// TIA Portal V15.1 export
// export: Created 2024-06-21T08:40:54.1245621Z, ExportSetting WithDefaults, DisplayName Totally Integrated Automation Portal, DisplayVersion V15.1 Update 5, DisplayName TIA Portal Openness, DisplayVersion V15.1 Update 5, DisplayName SINAMICS Startdrive Advanced, DisplayVersion V15.1, DisplayName G130, G150, S120, S150, SINAMICS MV, S210, DisplayVersion V15.1, DisplayName G110M, G120, G120C, G120D, G120P, DisplayVersion V15.1, DisplayName STEP 7 Professional, DisplayVersion V15.1 Update 5, DisplayName STEP 7 Safety, DisplayVersion V15.1, DisplayName WinCC Professional, DisplayVersion V15.1 Update 5, DisplayName SIMATIC Visualization Architect, DisplayVersion V15.1
FUNCTION "LBitToDword" : Void   // FC1027, FBD
TITLE = LBitToDWord
{ S7_Optimized_Access := 'TRUE' }
AUTHOR : VCC
FAMILY : Control
VERSION : 0.1
// =============================================================================
// Handles the conversion from bits to one DWord
// =============================================================================
// stored: AutoNumber false, IsIECCheckEnabled false, SetENOAutomatically False, UDAEnableTagReadback false
   VAR_INPUT
      I_0 : Bool;   // Alarm 00 / Input0
      I_1 : Bool;   // Alarm 01 / Input1
      I_2 : Bool;   // Alarm 02 / Input2
      I_3 : Bool;   // Alarm 03 / Input3
      I_4 : Bool;   // Alarm 04 / Input4
      I_5 : Bool;   // Alarm 05 / Input5
      I_6 : Bool;   // Alarm 06 / Input6
      I_7 : Bool;   // Alarm 07 / Input7
      I_8 : Bool;   // Alarm 08 / Input8
      I_9 : Bool;   // Alarm 09 / Input9
      I_10 : Bool;   // Alarm 10 / Input10
      I_11 : Bool;   // Alarm 11 / Input11
      I_12 : Bool;   // Alarm 12 / Input12
      I_13 : Bool;   // Alarm 13 / Input13
      I_14 : Bool;   // Alarm 14 / Input14
      I_15 : Bool;   // Alarm 15 / Input15
      I_16 : Bool;   // Alarm16 / Input16
      I_17 : Bool;   // Alarm17 / Input17
      I_18 : Bool;   // Alarm18 / Input18
      I_19 : Bool;   // Alarm19 / Input19
      I_20 : Bool;   // Alarm20 / Input20
      I_21 : Bool;   // Alarm21 / Input21
      I_22 : Bool;   // Alarm22 / Input22
      I_23 : Bool;   // Alarm23 / Input23
      I_24 : Bool;   // Alarm24 / Input24
      I_25 : Bool;   // Alarm25 / Input25
      I_26 : Bool;   // Alarm26 / Input26
      I_27 : Bool;   // Alarm27 / Input27
      I_28 : Bool;   // Alarm28 / Input28
      I_29 : Bool;   // Alarm29 / Input29
      I_30 : Bool;   // Alarm30 / Input30
      I_31 : Bool;   // Alarm31 / Input31
   END_VAR
   VAR_OUTPUT
      O_DWord : DWord;   // Alarn DWord for HMI / Dword Out
   END_VAR
BEGIN

REGION Network 1: Temp variable for HMI animation / **** 1 - Inputs **** Move Bit to temporary Word
   // Input
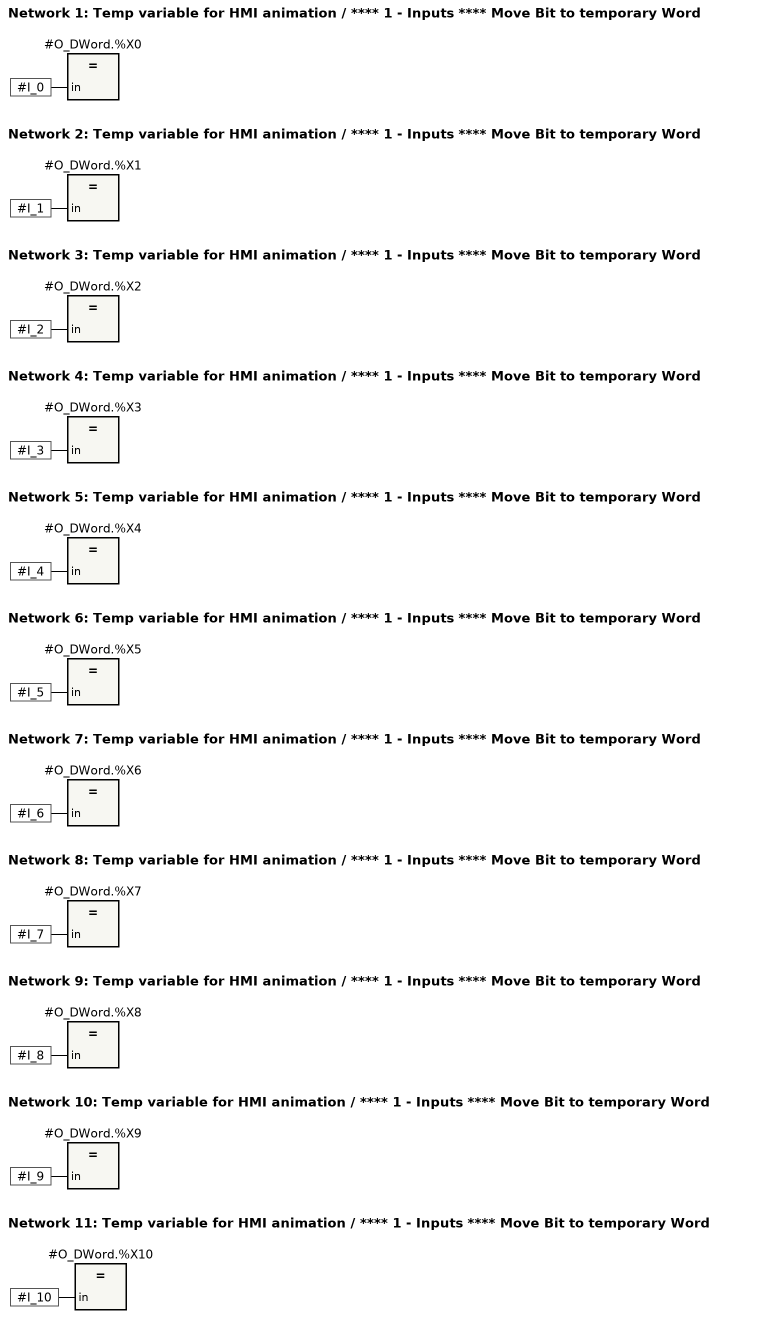
   #O_DWord.%X0 := #I_0;
END_REGION

REGION Network 2: Temp variable for HMI animation / **** 1 - Inputs **** Move Bit to temporary Word
   // Input
   #O_DWord.%X1 := #I_1;
END_REGION

REGION Network 3: Temp variable for HMI animation / **** 1 - Inputs **** Move Bit to temporary Word
   // Input
   #O_DWord.%X2 := #I_2;
END_REGION

REGION Network 4: Temp variable for HMI animation / **** 1 - Inputs **** Move Bit to temporary Word
   // Input
   #O_DWord.%X3 := #I_3;
END_REGION

REGION Network 5: Temp variable for HMI animation / **** 1 - Inputs **** Move Bit to temporary Word
   // Input
   #O_DWord.%X4 := #I_4;
END_REGION

REGION Network 6: Temp variable for HMI animation / **** 1 - Inputs **** Move Bit to temporary Word
   // Input
   #O_DWord.%X5 := #I_5;
END_REGION

REGION Network 7: Temp variable for HMI animation / **** 1 - Inputs **** Move Bit to temporary Word
   // Input
   #O_DWord.%X6 := #I_6;
END_REGION

REGION Network 8: Temp variable for HMI animation / **** 1 - Inputs **** Move Bit to temporary Word
   #O_DWord.%X7 := #I_7;
END_REGION

REGION Network 9: Temp variable for HMI animation / **** 1 - Inputs **** Move Bit to temporary Word
   // Input
   #O_DWord.%X8 := #I_8;
END_REGION

REGION Network 10: Temp variable for HMI animation / **** 1 - Inputs **** Move Bit to temporary Word
   // Input
   #O_DWord.%X9 := #I_9;
END_REGION

REGION Network 11: Temp variable for HMI animation / **** 1 - Inputs **** Move Bit to temporary Word
   // Input
   #O_DWord.%X10 := #I_10;
END_REGION

REGION Network 12: Temp variable for HMI animation / **** 1 - Inputs **** Move Bit to temporary Word
   // Input
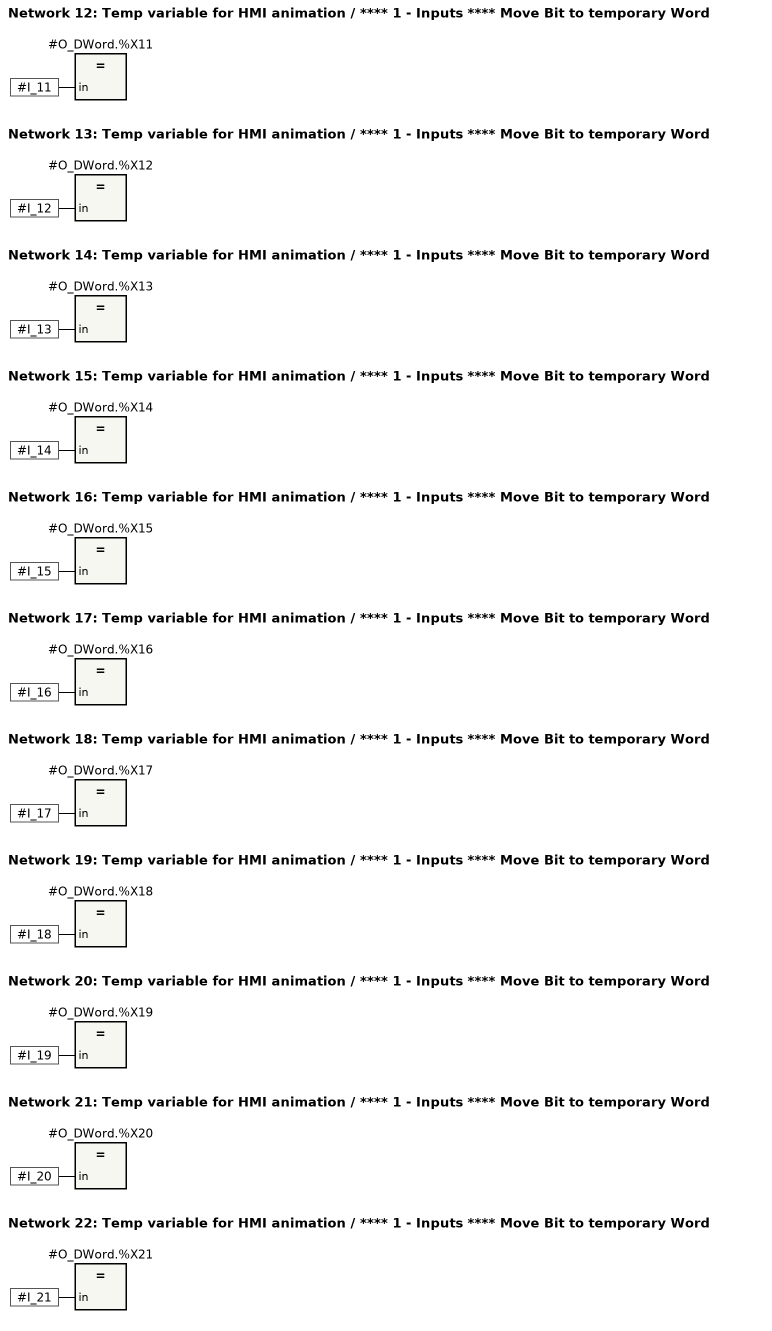
   #O_DWord.%X11 := #I_11;
END_REGION

REGION Network 13: Temp variable for HMI animation / **** 1 - Inputs **** Move Bit to temporary Word
   #O_DWord.%X12 := #I_12;
END_REGION

REGION Network 14: Temp variable for HMI animation / **** 1 - Inputs **** Move Bit to temporary Word
   // Input
   #O_DWord.%X13 := #I_13;
END_REGION

REGION Network 15: Temp variable for HMI animation / **** 1 - Inputs **** Move Bit to temporary Word
   // Input
   #O_DWord.%X14 := #I_14;
END_REGION

REGION Network 16: Temp variable for HMI animation / **** 1 - Inputs **** Move Bit to temporary Word
   // Input
   #O_DWord.%X15 := #I_15;
END_REGION

REGION Network 17: Temp variable for HMI animation / **** 1 - Inputs **** Move Bit to temporary Word
   #O_DWord.%X16 := #I_16;
END_REGION

REGION Network 18: Temp variable for HMI animation / **** 1 - Inputs **** Move Bit to temporary Word
   #O_DWord.%X17 := #I_17;
END_REGION

REGION Network 19: Temp variable for HMI animation / **** 1 - Inputs **** Move Bit to temporary Word
   // Input
   #O_DWord.%X18 := #I_18;
END_REGION

REGION Network 20: Temp variable for HMI animation / **** 1 - Inputs **** Move Bit to temporary Word
   // Input
   #O_DWord.%X19 := #I_19;
END_REGION

REGION Network 21: Temp variable for HMI animation / **** 1 - Inputs **** Move Bit to temporary Word
   // Input
   #O_DWord.%X20 := #I_20;
END_REGION

REGION Network 22: Temp variable for HMI animation / **** 1 - Inputs **** Move Bit to temporary Word
   // Input
   #O_DWord.%X21 := #I_21;
END_REGION

REGION Network 23: Temp variable for HMI animation / **** 1 - Inputs **** Move Bit to temporary Word
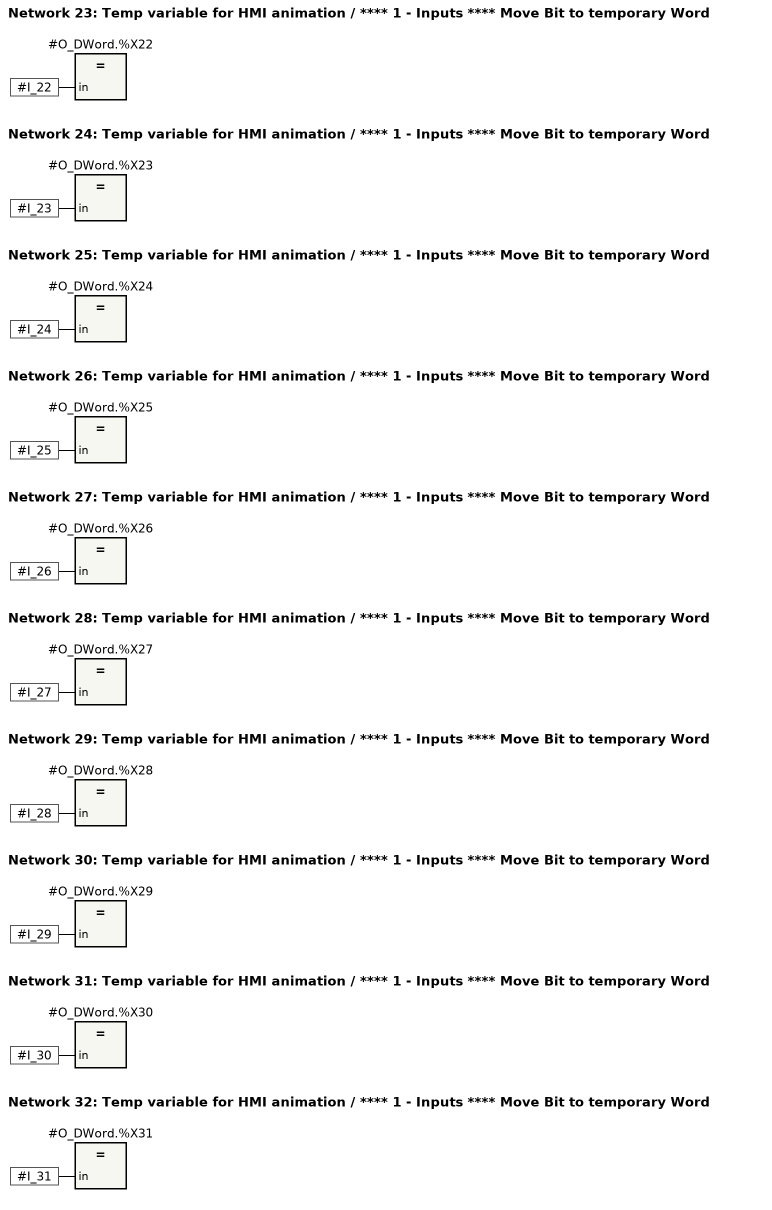
   #O_DWord.%X22 := #I_22;
END_REGION

REGION Network 24: Temp variable for HMI animation / **** 1 - Inputs **** Move Bit to temporary Word
   // Input
   #O_DWord.%X23 := #I_23;
END_REGION

REGION Network 25: Temp variable for HMI animation / **** 1 - Inputs **** Move Bit to temporary Word
   // Input
   #O_DWord.%X24 := #I_24;
END_REGION

REGION Network 26: Temp variable for HMI animation / **** 1 - Inputs **** Move Bit to temporary Word
   // Input
   #O_DWord.%X25 := #I_25;
END_REGION

REGION Network 27: Temp variable for HMI animation / **** 1 - Inputs **** Move Bit to temporary Word
   #O_DWord.%X26 := #I_26;
END_REGION

REGION Network 28: Temp variable for HMI animation / **** 1 - Inputs **** Move Bit to temporary Word
   #O_DWord.%X27 := #I_27;
END_REGION

REGION Network 29: Temp variable for HMI animation / **** 1 - Inputs **** Move Bit to temporary Word
   // Input
   #O_DWord.%X28 := #I_28;
END_REGION

REGION Network 30: Temp variable for HMI animation / **** 1 - Inputs **** Move Bit to temporary Word
   // Input
   #O_DWord.%X29 := #I_29;
END_REGION

REGION Network 31: Temp variable for HMI animation / **** 1 - Inputs **** Move Bit to temporary Word
   // Input
   #O_DWord.%X30 := #I_30;
END_REGION

REGION Network 32: Temp variable for HMI animation / **** 1 - Inputs **** Move Bit to temporary Word
   // Input
   #O_DWord.%X31 := #I_31;
END_REGION
END_FUNCTION
